// TIA Portal project "start-stop" (V16)

(* hardware
DEVICE "S7-1200 station_1"  S7-1200 Station
   slot 0: "Rack_0"  S7-1200 Rack  Rack  V1.0
   slot 1: "PLC_1"  CPU 1212C AC/DC/Rly  6ES7 212-1BE40-0XB0  V4.0
*)

// ===== PLC "PLC_1"  CPU 1212C AC/DC/Rly =====

VAR_GLOBAL   // PLC tag table "Default tag table"
   "start" AT %I0.1 : Bool;
   "stop" AT %I0.2 : Bool;
   "m2" AT %Q0.0 : Bool;
   "m3" AT %Q0.1 : Bool;
   "m1" AT %Q0.2 : Bool;
   "loop marker" AT %M0.0 : Bool;
   "t4 latch" AT %M0.1 : Bool;
   "M1 SS" AT %M0.2 : Bool;
   "M2 SS" AT %M0.3 : Bool;
   "M3 ss" AT %M0.4 : Bool;
END_VAR

// folder: System blocks/Program resources

DATA_BLOCK "T1"   // DB1
{ S7_Optimized_Access := 'TRUE' }
AUTHOR : Simatic
FAMILY : IEC
NAME : IEC_TMR
VERSION : 1.0
// stored: InstanceOfName IEC_TIMER
"IEC_TIMER"
BEGIN
END_DATA_BLOCK

DATA_BLOCK "T4"   // DB2
{ S7_Optimized_Access := 'TRUE' }
AUTHOR : Simatic
FAMILY : IEC
NAME : IEC_TMR
VERSION : 1.0
// stored: InstanceOfName IEC_TIMER
"IEC_TIMER"
BEGIN
END_DATA_BLOCK

DATA_BLOCK "T2"   // DB3
{ S7_Optimized_Access := 'TRUE' }
AUTHOR : Simatic
FAMILY : IEC
NAME : IEC_TMR
VERSION : 1.0
// stored: InstanceOfName IEC_TIMER
"IEC_TIMER"
BEGIN
END_DATA_BLOCK

DATA_BLOCK "T3"   // DB4
{ S7_Optimized_Access := 'TRUE' }
AUTHOR : Simatic
FAMILY : IEC
NAME : IEC_TMR
VERSION : 1.0
// stored: InstanceOfName IEC_TIMER
"IEC_TIMER"
BEGIN
END_DATA_BLOCK

// folder: (top level)

ORGANIZATION_BLOCK "Main"   // OB1, LAD, ProgramCycle
TITLE = "Main Program Sweep (Cycle)"
{ S7_Optimized_Access := 'TRUE' }
VERSION : 0.1
   VAR_INPUT
      Initial_Call : Bool;   // Initial call of this OB
      Remanence : Bool;   // =True, if remanent data are available
   END_VAR
BEGIN

REGION Network 1
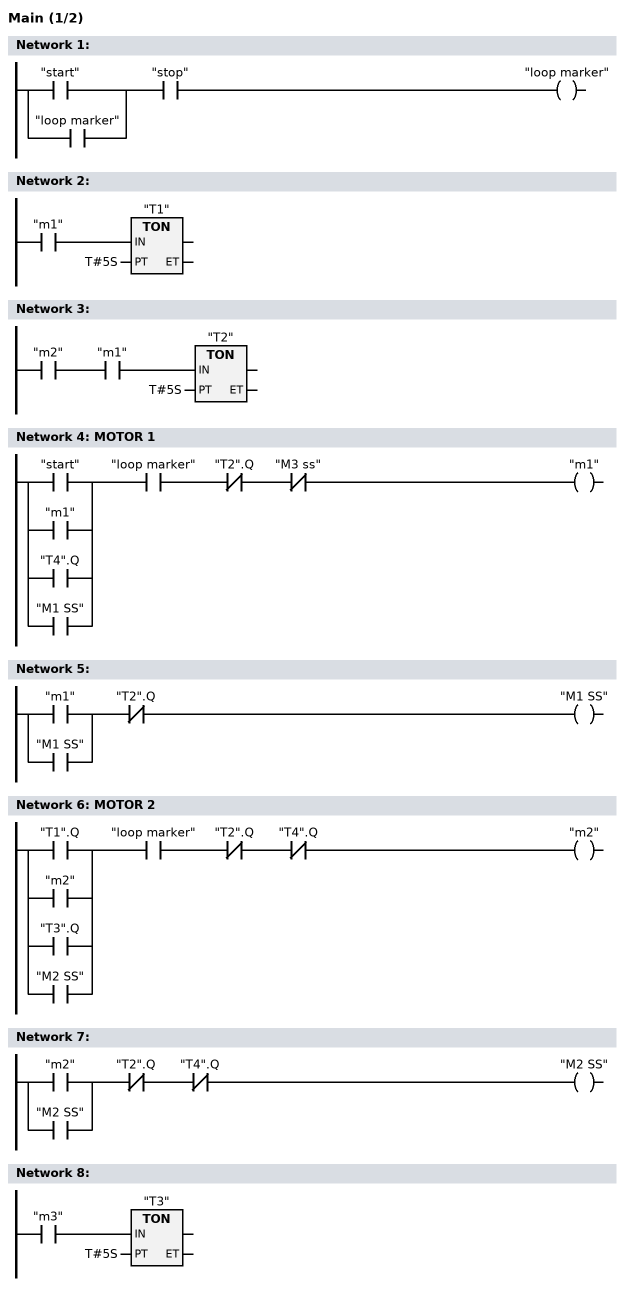
   RUNG wire#powerrail
      Contact( "start" )
      wire#w1
      Contact( "stop" )
      Coil( "loop marker" )
   END_RUNG
   RUNG wire#powerrail
      Contact( "loop marker" )
   END_RUNG wire#w1
   // the same network as SCL:
   "loop marker" := ("start" OR "loop marker") AND "stop";
END_REGION

REGION Network 2
   "T1".TON(IN := "m1", PT := T#5S);
END_REGION

REGION Network 3
   "T2".TON(IN := "m2" AND "m1", PT := T#5S);
END_REGION

REGION Network 4: MOTOR 1
   RUNG wire#powerrail
      Contact( "start" )
      wire#w1
      Contact( "loop marker" )
      I_Contact( "T2".Q )
      I_Contact( "M3 ss" )
      Coil( "m1" )
   END_RUNG
   RUNG wire#powerrail
      Contact( "m1" )
   END_RUNG wire#w1
   RUNG wire#powerrail
      Contact( "T4".Q )
   END_RUNG wire#w1
   RUNG wire#powerrail
      Contact( "M1 SS" )
   END_RUNG wire#w1
   // the same network as SCL:
   "m1" := ("start" OR "m1" OR "T4".Q OR "M1 SS") AND "loop marker" AND NOT "T2".Q AND NOT "M3 ss";
END_REGION

REGION Network 5
   RUNG wire#powerrail
      Contact( "m1" )
      wire#w1
      I_Contact( "T2".Q )
      Coil( "M1 SS" )
   END_RUNG
   RUNG wire#powerrail
      Contact( "M1 SS" )
   END_RUNG wire#w1
   // the same network as SCL:
   "M1 SS" := ("m1" OR "M1 SS") AND NOT "T2".Q;
END_REGION

REGION Network 6: MOTOR 2
   RUNG wire#powerrail
      Contact( "T1".Q )
      wire#w1
      Contact( "loop marker" )
      I_Contact( "T2".Q )
      I_Contact( "T4".Q )
      Coil( "m2" )
   END_RUNG
   RUNG wire#powerrail
      Contact( "m2" )
   END_RUNG wire#w1
   RUNG wire#powerrail
      Contact( "T3".Q )
   END_RUNG wire#w1
   RUNG wire#powerrail
      Contact( "M2 SS" )
   END_RUNG wire#w1
   // the same network as SCL:
   "m2" := ("T1".Q OR "m2" OR "T3".Q OR "M2 SS") AND "loop marker" AND NOT "T2".Q AND NOT "T4".Q;
END_REGION

REGION Network 7
   RUNG wire#powerrail
      Contact( "m2" )
      wire#w1
      I_Contact( "T2".Q )
      I_Contact( "T4".Q )
      Coil( "M2 SS" )
   END_RUNG
   RUNG wire#powerrail
      Contact( "M2 SS" )
   END_RUNG wire#w1
   // the same network as SCL:
   "M2 SS" := ("m2" OR "M2 SS") AND NOT "T2".Q AND NOT "T4".Q;
END_REGION

REGION Network 8
   "T3".TON(IN := "m3", PT := T#5S);
END_REGION

REGION Network 9: MOTOR 3
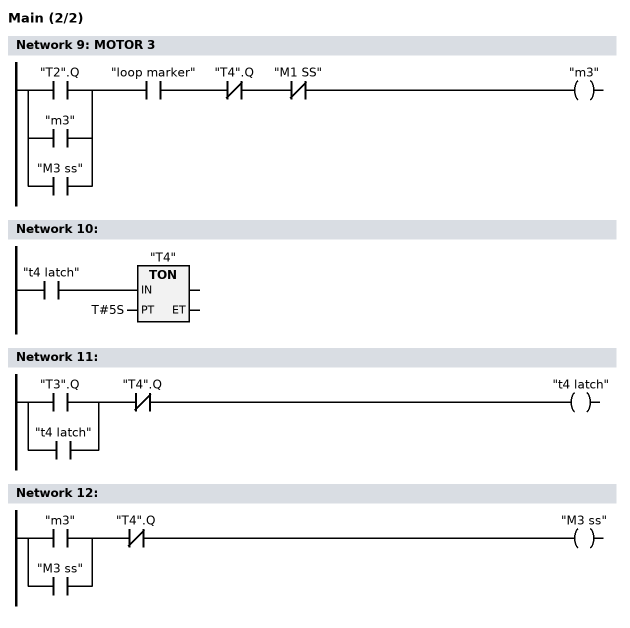
   RUNG wire#powerrail
      Contact( "T2".Q )
      wire#w1
      Contact( "loop marker" )
      I_Contact( "T4".Q )
      I_Contact( "M1 SS" )
      Coil( "m3" )
   END_RUNG
   RUNG wire#powerrail
      Contact( "m3" )
   END_RUNG wire#w1
   RUNG wire#powerrail
      Contact( "M3 ss" )
   END_RUNG wire#w1
   // the same network as SCL:
   "m3" := ("T2".Q OR "m3" OR "M3 ss") AND "loop marker" AND NOT "T4".Q AND NOT "M1 SS";
END_REGION

REGION Network 10
   "T4".TON(IN := "t4 latch", PT := T#5S);
END_REGION

REGION Network 11
   RUNG wire#powerrail
      Contact( "T3".Q )
      wire#w1
      I_Contact( "T4".Q )
      Coil( "t4 latch" )
   END_RUNG
   RUNG wire#powerrail
      Contact( "t4 latch" )
   END_RUNG wire#w1
   // the same network as SCL:
   "t4 latch" := ("T3".Q OR "t4 latch") AND NOT "T4".Q;
END_REGION

REGION Network 12
   RUNG wire#powerrail
      Contact( "m3" )
      wire#w1
      I_Contact( "T4".Q )
      Coil( "M3 ss" )
   END_RUNG
   RUNG wire#powerrail
      Contact( "M3 ss" )
   END_RUNG wire#w1
   // the same network as SCL:
   "M3 ss" := ("m3" OR "M3 ss") AND NOT "T4".Q;
END_REGION
END_ORGANIZATION_BLOCK